% RSLogix 500 project micrologix1000_program.RSS, saved by version 8.40.00.08 %
PROJECT "PRESS64"    % processor: MicroLogix 1000 %

PROGRAM FILES
  LAD 2 "MAIN_PROG"  26 rungs
  LAD 3 "USER_FAULT"  1 rungs
  LAD 4 "HSC_INT"  1 rungs
  LAD 5 "STI_INT"  1 rungs
  LAD 6, 7, 8, 9, 10, 11, 12, 13, 14, 15, 16: only END

DATA FILES
  O0 OUTPUT  1 elements
  I1 INPUT  2 elements
  S2 STATUS  33 elements
  B3 BINARY  32 elements
  T4 TIMER  40 elements
  C5 COUNTER  32 elements
  R6 CONTROL  16 elements
  N7 INTEGER  105 elements

LADDER 2 "MAIN_PROG"
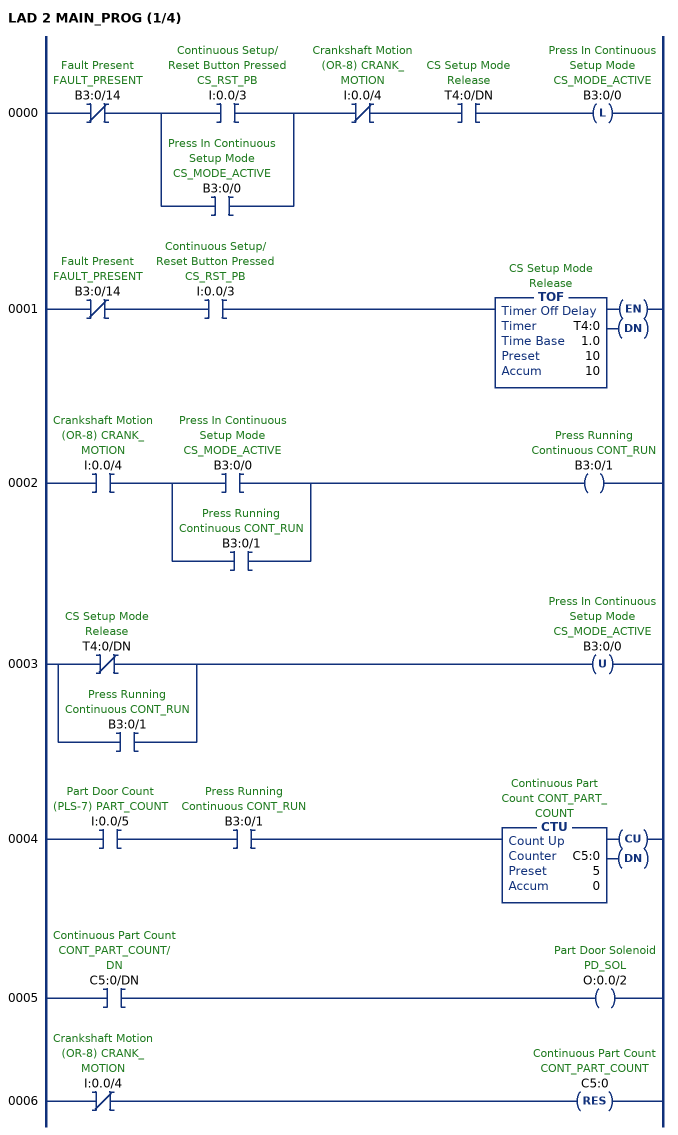
% Rung: 0 %
SOR XIO B3:0/14 BST XIC I:0.0/3 NXB XIC B3:0/0 BND XIO I:0.0/4 XIC T4:0/DN OTL B3:0/0 EOR
%   B3:0/14  FAULT_PRESENT  "Fault Present" %
%   I:0.0/3  CS_RST_PB  "Continuous Setup/ Reset Button Pressed" %
%   B3:0/0  CS_MODE_ACTIVE  "Press In Continuous Setup Mode" %
%   I:0.0/4  CRANK_MOTION  "Crankshaft Motion (OR-8)" %
%   T4:0  "CS Setup Mode Release" %
% Rung: 1 %
SOR XIO B3:0/14 XIC I:0.0/3 TOF T4:0 1.0 10 10 EOR
%   B3:0/14  FAULT_PRESENT  "Fault Present" %
%   I:0.0/3  CS_RST_PB  "Continuous Setup/ Reset Button Pressed" %
%   T4:0  "CS Setup Mode Release" %
% Rung: 2 %
SOR XIC I:0.0/4 BST XIC B3:0/0 NXB XIC B3:0/1 BND OTE B3:0/1 EOR
%   I:0.0/4  CRANK_MOTION  "Crankshaft Motion (OR-8)" %
%   B3:0/0  CS_MODE_ACTIVE  "Press In Continuous Setup Mode" %
%   B3:0/1  CONT_RUN  "Press Running Continuous" %
% Rung: 3 %
SOR BST XIO T4:0/DN NXB XIC B3:0/1 BND OTU B3:0/0 EOR
%   T4:0  "CS Setup Mode Release" %
%   B3:0/1  CONT_RUN  "Press Running Continuous" %
%   B3:0/0  CS_MODE_ACTIVE  "Press In Continuous Setup Mode" %
% Rung: 4 %
SOR XIC I:0.0/5 XIC B3:0/1 CTU C5:0 5 0 EOR
%   I:0.0/5  PART_COUNT  "Part Door Count (PLS-7)" %
%   B3:0/1  CONT_RUN  "Press Running Continuous" %
%   C5:0  CONT_PART_COUNT  "Continuous Part Count" %
% Rung: 5 %
SOR XIC C5:0/DN OTE O:0.0/2 EOR
%   C5:0  CONT_PART_COUNT  "Continuous Part Count" %
%   O:0.0/2  PD_SOL  "Part Door Solenoid" %
% Rung: 6 %
SOR XIO I:0.0/4 RES C5:0 EOR
%   I:0.0/4  CRANK_MOTION  "Crankshaft Motion (OR-8)" %
%   C5:0  CONT_PART_COUNT  "Continuous Part Count" %

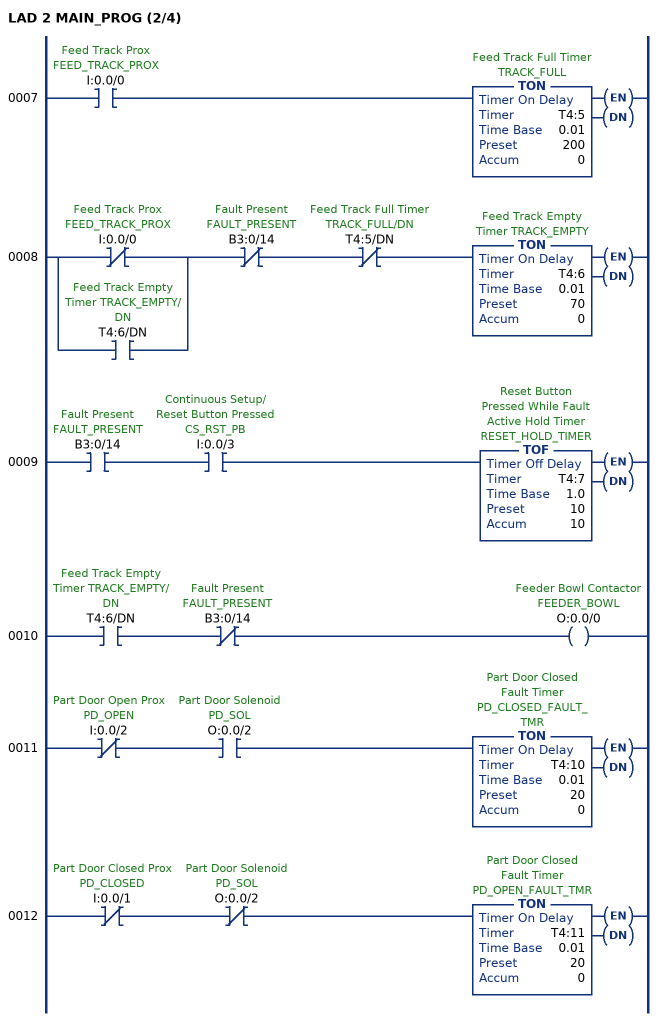
% Rung: 7 %
SOR XIC I:0.0/0 TON T4:5 0.01 200 0 EOR
%   I:0.0/0  FEED_TRACK_PROX  "Feed Track Prox" %
%   T4:5  TRACK_FULL  "Feed Track Full Timer" %
% Rung: 8 %
SOR BST XIO I:0.0/0 NXB XIC T4:6/DN BND XIO B3:0/14 XIO T4:5/DN TON T4:6 0.01 70 0 EOR
%   I:0.0/0  FEED_TRACK_PROX  "Feed Track Prox" %
%   T4:6  TRACK_EMPTY  "Feed Track Empty Timer" %
%   B3:0/14  FAULT_PRESENT  "Fault Present" %
%   T4:5  TRACK_FULL  "Feed Track Full Timer" %
% Rung: 9 %
SOR XIC B3:0/14 XIC I:0.0/3 TOF T4:7 1.0 10 10 EOR
%   B3:0/14  FAULT_PRESENT  "Fault Present" %
%   I:0.0/3  CS_RST_PB  "Continuous Setup/ Reset Button Pressed" %
%   T4:7  RESET_HOLD_TIMER  "Reset Button Pressed While Fault Active Hold Timer" %
% Rung: 10 %
SOR XIC T4:6/DN XIO B3:0/14 OTE O:0.0/0 EOR
%   T4:6  TRACK_EMPTY  "Feed Track Empty Timer" %
%   B3:0/14  FAULT_PRESENT  "Fault Present" %
%   O:0.0/0  FEEDER_BOWL  "Feeder Bowl Contactor" %
% Rung: 11 %
SOR XIO I:0.0/2 XIC O:0.0/2 TON T4:10 0.01 20 0 EOR
%   I:0.0/2  PD_OPEN  "Part Door Open Prox" %
%   O:0.0/2  PD_SOL  "Part Door Solenoid" %
%   T4:10  PD_CLOSED_FAULT_TMR  "Part Door Closed Fault Timer" %
% Rung: 12 %
SOR XIO I:0.0/1 XIO O:0.0/2 TON T4:11 0.01 20 0 EOR
%   I:0.0/1  PD_CLOSED  "Part Door Closed Prox" %
%   O:0.0/2  PD_SOL  "Part Door Solenoid" %
%   T4:11  PD_OPEN_FAULT_TMR  "Part Door Closed Fault Timer" %

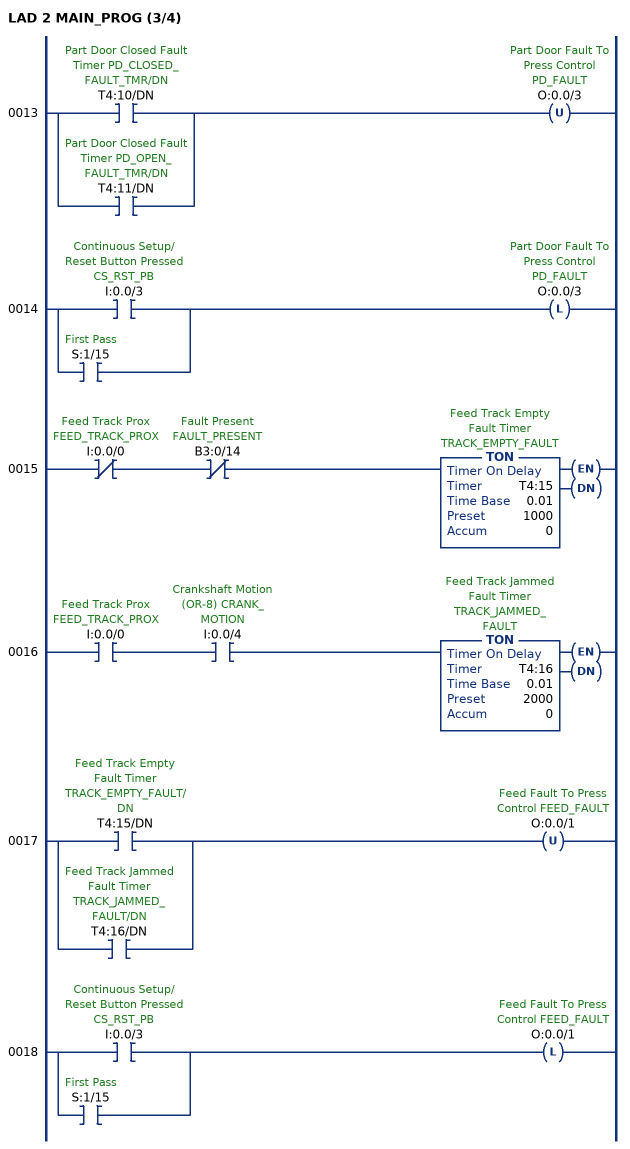
% Rung: 13 %
SOR BST XIC T4:10/DN NXB XIC T4:11/DN BND OTU O:0.0/3 EOR
%   T4:10  PD_CLOSED_FAULT_TMR  "Part Door Closed Fault Timer" %
%   T4:11  PD_OPEN_FAULT_TMR  "Part Door Closed Fault Timer" %
%   O:0.0/3  PD_FAULT  "Part Door Fault To Press Control" %
% Rung: 14 %
SOR BST XIC I:0.0/3 NXB XIC S:1/15 BND OTL O:0.0/3 EOR
%   I:0.0/3  CS_RST_PB  "Continuous Setup/ Reset Button Pressed" %
%   S:1/15  "First Pass" %
%   O:0.0/3  PD_FAULT  "Part Door Fault To Press Control" %
% Rung: 15 %
SOR XIO I:0.0/0 XIO B3:0/14 TON T4:15 0.01 1000 0 EOR
%   I:0.0/0  FEED_TRACK_PROX  "Feed Track Prox" %
%   B3:0/14  FAULT_PRESENT  "Fault Present" %
%   T4:15  TRACK_EMPTY_FAULT  "Feed Track Empty Fault Timer" %
% Rung: 16 %
SOR XIC I:0.0/0 XIC I:0.0/4 TON T4:16 0.01 2000 0 EOR
%   I:0.0/0  FEED_TRACK_PROX  "Feed Track Prox" %
%   I:0.0/4  CRANK_MOTION  "Crankshaft Motion (OR-8)" %
%   T4:16  TRACK_JAMMED_FAULT  "Feed Track Jammed Fault Timer" %
% Rung: 17 %
SOR BST XIC T4:15/DN NXB XIC T4:16/DN BND OTU O:0.0/1 EOR
%   T4:15  TRACK_EMPTY_FAULT  "Feed Track Empty Fault Timer" %
%   T4:16  TRACK_JAMMED_FAULT  "Feed Track Jammed Fault Timer" %
%   O:0.0/1  FEED_FAULT  "Feed Fault To Press Control" %
% Rung: 18 %
SOR BST XIC I:0.0/3 NXB XIC S:1/15 BND OTL O:0.0/1 EOR
%   I:0.0/3  CS_RST_PB  "Continuous Setup/ Reset Button Pressed" %
%   S:1/15  "First Pass" %
%   O:0.0/1  FEED_FAULT  "Feed Fault To Press Control" %

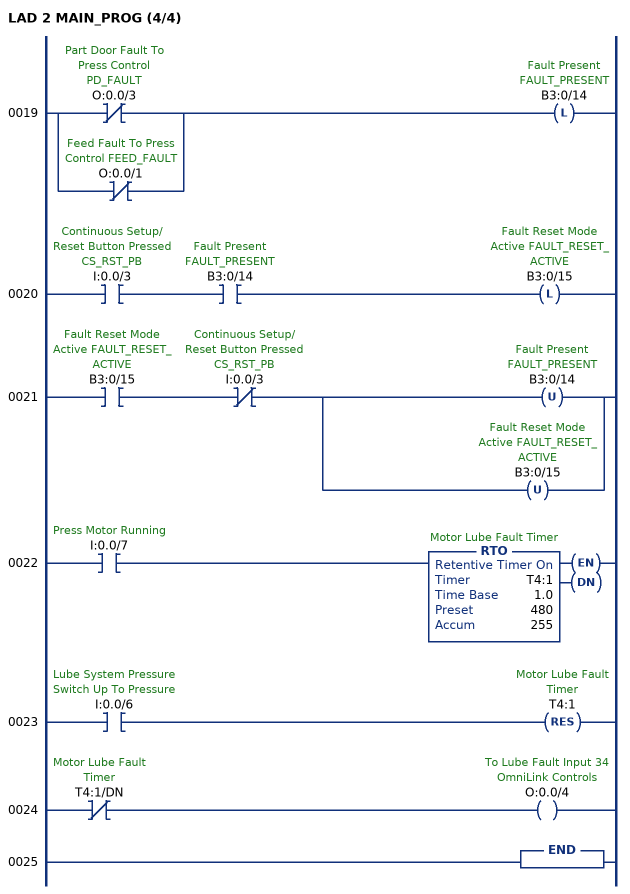
% Rung: 19 %
SOR BST XIO O:0.0/3 NXB XIO O:0.0/1 BND OTL B3:0/14 EOR
%   O:0.0/3  PD_FAULT  "Part Door Fault To Press Control" %
%   O:0.0/1  FEED_FAULT  "Feed Fault To Press Control" %
%   B3:0/14  FAULT_PRESENT  "Fault Present" %
% Rung: 20 %
SOR XIC I:0.0/3 XIC B3:0/14 OTL B3:0/15 EOR
%   I:0.0/3  CS_RST_PB  "Continuous Setup/ Reset Button Pressed" %
%   B3:0/14  FAULT_PRESENT  "Fault Present" %
%   B3:0/15  FAULT_RESET_ACTIVE  "Fault Reset Mode Active" %
% Rung: 21 %
SOR XIC B3:0/15 XIO I:0.0/3 BST OTU B3:0/14 NXB OTU B3:0/15 BND EOR
%   B3:0/15  FAULT_RESET_ACTIVE  "Fault Reset Mode Active" %
%   I:0.0/3  CS_RST_PB  "Continuous Setup/ Reset Button Pressed" %
%   B3:0/14  FAULT_PRESENT  "Fault Present" %
% Rung: 22 %
SOR XIC I:0.0/7 RTO T4:1 1.0 480 255 EOR
%   I:0.0/7  "Press Motor Running" %
%   T4:1  "Motor Lube Fault Timer" %
% Rung: 23 %
SOR XIC I:0.0/6 RES T4:1 EOR
%   I:0.0/6  "Lube System Pressure Switch Up To Pressure" %
%   T4:1  "Motor Lube Fault Timer" %
% Rung: 24 %
SOR XIO T4:1/DN OTE O:0.0/4 EOR
%   T4:1  "Motor Lube Fault Timer" %
%   O:0.0/4  "To Lube Fault Input 34 OmniLink Controls" %
% Rung: 25 %
SOR END EOR

OTHER DOCUMENTED ADDRESSES
  DFILE:0  "OUTPUT"
  DFILE:1  "INPUT"
  DFILE:2  "STATUS"
  DFILE:3  "BINARY"
  DFILE:4  "TIMER"
  DFILE:5  "COUNTER"
  DFILE:6  "CONTROL"
  DFILE:7  "INTEGER"
  DFILE:8  "FLOAT"

DATA TABLE (non-zero values as saved)
DATA B3
% B3:0 % 0X4000 0X0000 0X0000 0X0000 0X0000 0X0000 0X0000 0X0000 0X0000 0X0000
DATA T4
% .PRE .ACC %
% T4:0 % 10 10
% T4:1 % 480 255
% T4:5 % 200 0
% T4:6 % 70 0
% T4:7 % 10 10
% T4:10 % 20 0
% T4:11 % 20 0
% T4:15 % 1000 0
% T4:16 % 2000 0
DATA C5
% .PRE .ACC %
% C5:0 % 5 0
